(* PLC project testTypes *)
(* stored: creationDateTime 2018-01-30T20:16:00, modificationDateTime 2018-01-30T20:16:00 *)

TYPE digitalSignal : BOOL := false;
END_TYPE

TYPE commandOnOff : BOOL;
END_TYPE

TYPE absoluteTemperature : REAL := 273.16;
END_TYPE

TYPE degreesFahrenheit : absoluteTemperature;
END_TYPE

TYPE trafficLightStates : (red, yellow, green);
END_TYPE

TYPE machineStates : (idle, busy, service);
END_TYPE

TYPE commStates : (idle := 0, msg_detected, msg_sent := 5);
END_TYPE

TYPE analogValue : UINT(0..27648) := 13824;
END_TYPE

TYPE floorNumber : SINT(-5..50);
END_TYPE

TYPE switchData : STRUCT
  Open : BOOL;
  Closed : BOOL;
  Measurements : STRUCT
    Voltage : REAL;
    Current : REAL;
  END_STRUCT;
END_STRUCT;
END_TYPE

TYPE realArray : ARRAY[0..5, -3..12] OF REAL;
END_TYPE

FUNCTION signal : BOOL
  VAR_INPUT  (* input *)
    in : in;
  END_VAR
  VAR_INPUT  (* input *)
    on : on;
  END_VAR

END_FUNCTION

FUNCTION escalator
  VAR_INPUT  (* Input *)
    up : INT := 1;
  END_VAR
  VAR  (* local *)
    first : INT;
    second : INT := 2;
    third : INT := 3;
  END_VAR
  VAR_OUTPUT  (* output *)
    down : INT;
  END_VAR

END_FUNCTION

FUNCTION light
  VAR_INPUT  (* inPut *)
    lighton : BOOL := true;
  END_VAR
  VAR_INPUT  (* INput *)
    lightof : BOOL := false;
  END_VAR
  VAR_TEMP  (* TEMP *)
    colour : LWORD;
  END_VAR

END_FUNCTION

FUNCTION door : TIME
  VAR_IN_OUT  (* inout *)
    open : TIME;
  END_VAR
  VAR_OUTPUT  (* output *)
    close : TIME;
  END_VAR

END_FUNCTION

FUNCTION open
  VAR  (* LOcal *)
    turnon : INT := 1;
    turnoff : INT := 0;
  END_VAR
  VAR_TEMP  (* TeMp *)
    close : INT;
  END_VAR

END_FUNCTION

FUNCTION_BLOCK value

END_FUNCTION_BLOCK

PROGRAM start

END_PROGRAM

FUNCTION distance : kilometers

END_FUNCTION

FUNCTION time : TIME

END_FUNCTION

FUNCTION elevator : INT
  VAR  (* floor *)
    first : REAL;
    second : REAL;
    third : REAL;
    fourth : REAL;
  END_VAR

END_FUNCTION

FUNCTION aircondition
  VAR_OUTPUT  (* output *)
    start : INT := 28;
  END_VAR
  VAR_OUTPUT  (* OutPut= *)
    temprature : REAL := 32.5;
  END_VAR
  VAR_TEMP  (* temP *)
    measurment : REAL;
  END_VAR

END_FUNCTION

FUNCTION window
  VAR_IN_OUT  (* inout *)
    close : TIME;
  END_VAR

END_FUNCTION

FUNCTION engine
  VAR_INPUT  (* input *)
    var : BOOL;
  END_VAR
  VAR  (* Local *)
    start : BYTE;
    pause : BYTE;
    stop : BYTE;
  END_VAR

END_FUNCTION

PROGRAM trafficLight

END_PROGRAM

FUNCTION degreesFahrenheit : absoluteTemperature
  VAR_INPUT  (* input *)
    temperature : absoluteTemperature;
  END_VAR
  VAR_TEMP  (* Temp *)
    Temperature : LREAL;
  END_VAR
  VAR_IN_OUT  (* inOut *)
    temp : LREAL;
  END_VAR

END_FUNCTION

CONFIGURATION conf1
  RESOURCE res1 ON PLC
  END_RESOURCE
END_CONFIGURATION
